PROGRAM P_Demo_FB_DMXSetResetDevice
VAR
    fbResetDevice     : FB_DMXSetResetDevice;         // 远程复位单台设备
    stDmxCmdBuffer    : ST_DMXCommandBuffer;          // 与通讯 FB 共用
    wTargetManufId    : WORD := 16#4241;              // 目标灯具厂商 ID
    dwTargetDeviceId  : DWORD := 16#12131415;         // 目标灯具设备 ID
    byTargetPort      : BYTE := 0;                    // 根设备通道 0
    eResetKind        : E_DMXResetDeviceType := eDMXResetDeviceTypeWarm;  // 热复位
    bDoReset          : BOOL := FALSE;                // 在线给一次上升沿触发
    bBusy             : BOOL;
    bError            : BOOL;
    udiErrId          : UDINT;
END_VAR

// ============================================================
// Tc2_DMX.FB_DMXSetResetDevice 演示程序
// ============================================================
// 场景：某盏灯通讯异常但物理可达，不派人现场断电，直接从 PLC 远程复位恢复。
// 价值：把远程重启单台设备做成一次调用，省去派人到现场或整段总线断电。
// 验证：给 bDoReset 一次上升沿（eResetKind=eDMXResetDeviceTypeWarm）-> bBusy 短暂 TRUE -> 回 FALSE 后目标设备应短时离线再恢复；若 bError 且 udiErrId=0x8007 说明复位类型越界。
// 验证步骤：
//   1. 右键 PLC 项目下 POUs 文件夹 → Add → Existing Item → 选本 .TcPOU 文件
//   2. 引用 Tc2_DMX；同项目里放一个 FB_EL6851CommunicationEx 实例并共用 stDmxCmdBuffer（非 CycleMode）
//   3. 编译 → 登录 → 运行；按上方『验证』行在线给上升沿观察
// ============================================================

fbResetDevice(
    bStart                     := bDoReset,
    wDestinationManufacturerId := wTargetManufId,
    dwDestinationDeviceId      := dwTargetDeviceId,
    byPortId                   := byTargetPort,
    eResetDeviceType           := eResetKind,
    dwOptions                  := 0,
    stCommandBuffer            := stDmxCmdBuffer,
    bBusy                      => bBusy,
    bError                     => bError,
    udiErrorId                 => udiErrId
);

END_PROGRAM

(* stored: Version 1.1.0.1, ProductVersion 3.1.4024.5
   POU P_Demo_FB_DMXSetResetDevice: Id {c0b7af7c-c40a-5598-bd85-ac80e8966618}, SpecialFunc None *)
